Fanuc KAREL source: kx00019.KL

PROGRAM KX00019
%STACKSIZE=65535
%PRIORITY=65535
%NOLOCKGROUP
VAR
I : INTEGER
J : INTEGER
B : BOOLEAN
F : FILE
S : STRING[80]
P : XYZWPR
-- UNRESOLVED DECLARATIONS (source type spelling not recovered)
-- SH : ARRAY[4] OF TYPE_0x0017 (type_u16=0x2017)
BEGIN
-- UNRESOLVED_PC line 12 opcodes [2E 22 9D 33 B4] marker_code=0
-- UNRESOLVED_PC line 13 opcodes [22 9D 33 B3 23] marker_code=19
END KX00019
